Fanuc KAREL source: kt00604.KL

-- PROVISIONAL review KL for V940-1; original PC SHA256 9907d5bfae8d429ca779416f01524d1c0583180a699cf4f51ce2372b1f3ec46c
-- Incomplete behavior may be omitted. Consult companion uncertainty JSON. Do not deploy.
PROGRAM KT00604
%NOLOCKGROUP
VAR
  I1 : INTEGER
  I2 : INTEGER
  OUT : INTEGER
BEGIN
  -- V9_ZERO_TABLE_METADATA_HINT layout=0001; no indexed target words; source/name/runtime held
  -- UNRESOLVED_PC offsets 5-16; opcodes 2E,23
  -- UNRESOLVED_PC offsets 21-32; opcodes 2E,23
  -- UNRESOLVED_PC offsets 37-48; opcodes 2E,23
  -- UNRESOLVED_PC offsets 53-64; opcodes 2E,23
  -- UNRESOLVED_PC offsets 69-82; opcodes 21,51,23
  -- UNRESOLVED_PC offsets 87-91; opcodes 7F
END KT00604
